FUNCTION UpdateEventWithSystemTime 
VAR_INPUT
	stEvent : REFERENCE TO ST_Event;
END_VAR
VAR
	fbGETSYSTEMTIME : GETSYSTEMTIME;
	stFileTime: T_FILETIME;
	
END_VAR

fbGETSYSTEMTIME( timeLoDW => stFileTime.dwLowDateTime,
	              timeHiDW => stFileTime.dwHighDateTime);


stEvent.dtTimestamp := FILETIME_TO_DT(fileTime := stFileTime);

END_FUNCTION

(* stored: Version 1.1.0.1, ProductVersion 3.1.4024.12
   POU UpdateEventWithSystemTime: Id {7b248580-b99c-4232-8aaf-016fef871369}, SpecialFunc None *)
